{attribute addProperty BoxType "EJ1957-0000-0017"}
{attribute addProperty Id "FSLOGIC_InputsFSLOGIC_Inputs_8BA5C933162FSLOGIC_OutputsEMPTY_STRUCTURE00"}
{attribute addProperty CRC "1046630713"}
{attribute addProperty SizeInBites "16"}
{attribute addProperty SizeInBytes "2"}
TYPE Module_4_FSLOGIC_3E625139 :
STRUCT
	{attribute addProperty Name "FSLOGIC_Inputs"}
	FSLOGIC_Inputs  : FSLOGIC_Inputs_8BA5C933;
	{attribute addProperty Name "FSLOGIC_Outputs"}
	FSLOGIC_Outputs  : EMPTY_STRUCTURE;
END_STRUCT
END_TYPE

(* stored: Version 1.2.0.0, ProductVersion 3.1.4024.9
   DUT Module_4_FSLOGIC_3E625139: Id {2f8a8fff-5bec-4124-9387-f6da53628f4c} *)
